FUNCTION_BLOCK FB_ServoVise
VAR_INPUT
	bErrorAck				: BOOL;
	bEnable					: BOOL;
	eCommand				: E_ServoVise_Command;
	bManualMode				: BOOL;
	lrTargetDistance		: LREAL;			// [mm]		Target distance without torque limit
	lrVisePosition			: LREAL;			// [mm]		Value of distance sensor
	bVisePosValid			: BOOL;				// []		Distane sensor status
	nTargetVelocity			: LREAL;			// [mm/s]
	nTorque					: LREAL := 20.0;	// [Nm]
	nTorqueRamp				: LREAL := 10.0;	// [%/s]
	nTorqueVelocityLimit	: LREAL := 0.1;		// [mm/s]
	nOverride				: LREAL := 100.0;	// [%] 
	nAttachVelocity			: LREAL := 0.1;
	nCalOffset_1			: LREAL := 22.32;
	nCalOffset_2			: LREAL := 99.01;
	nOpenOffset				: LREAL := 4;
	eViseJawState			: E_ViseJawState := E_ViseJawState.P1_0_120;
	stAxisEvent				: TcEventEntry;	(*Event definition*)
END_VAR
VAR_OUTPUT
	bReady					: BOOL;
	bBusy 					: BOOL;
	bDone 					: BOOL;
	bError 					: BOOL;
END_VAR
VAR (* Drive *)
	Axis					: AXIS_REF;
	fbPower					: MC_Power;
	fbMoveRelative			: MC_MoveRelative;
	fbReadDriveOpMode		: MC_ReadDriveOperationMode;
	fbWriteDriveOpMode		: MC_WriteDriveOperationMode;
	fbStop					: MC_Halt;
	fbHalt					: MC_Stop;
	fbTorqueControl			: MC_TorqueControl;	
	fbJog					: MC_Jog;
	fbTorqueCheck			: FB_TorqueCheck;	

	fbSoEReset				: FB_SoEReset;
	fbReset					: MC_Reset;
END_VAR
VAR (* State control *)
	nState 					: UDINT;
	nLastState				: UDINT;
	sState					: STRING;
	nTorqueRelief			: LREAL := 0.005;	// 0.005mm = 0.9°
	
	// Error control
	bIsInitalized			: BOOL;
	fbAlarm					: FB_TcAlarm;
	nGlobalAxisErrorID		: UDINT;
	
	//LastStates
	anLastStates			: ARRAY[0..500] OF UDINT;
    iLastStates				: INT;
	nRealVisePos			: LREAL;
END_VAR
VAR CONSTANT									//																			%     Tmax    i   Theta															
	nTScale					: LREAL := 2.3923;	// nTorque[Nm] / nTScale[Nm/%] = Required_torque_value[%]		{nTScale = 0.01 * 5.09 * 50 * 0.94}
END_VAR

(* Timers **************************************)

(* Enable **************************************)
IF NOT bEnable THEN
	fbPower.Enable := FALSE;
	fbTorqueControl.Execute := FALSE;
	fbMoveRelative.Execute := FALSE;
	nState := 0;
END_IF

(* States **************************************)
IF nLastState <> nState THEN
	nLastState := nState;
END_IF

(* State history ************************************************)
IF(nState >= 100) AND (nState <= 20000) THEN
(*Steps before any state*)
	IF anLastStates[0] <> nState THEN
		FOR iLastStates:=500 TO 1 BY -1 DO
			anLastStates[iLastStates]:= anLastStates[iLastStates-1];
		END_FOR
		anLastStates[0]:= nState;
	END_IF
END_IF	

(* Manual mode **************************************)
IF bManualMode THEN
	nState := 150000;
END_IF

(*Calculate Vise position **************************************)
IF eViseJawState = E_ViseJawState.P1_0_120 THEN
	nRealVisePos := lrVisePosition + nCalOffset_1;
ELSE
	nRealVisePos := lrVisePosition + nCalOffset_2;
END_IF

(* Error handling Tc3_EventLogger *******************************)
IF NOT bIsInitalized THEN
	bIsInitalized  :=  TRUE;
	fbAlarm.CreateEx(stAxisEvent, TRUE, 0);
END_IF

(* Error acknoledge **************************************)
IF bErrorAck THEN
	IF fbAlarm.eConfirmationState = 2 THEN
		fbAlarm.Confirm(0);
	END_IF
END_IF

IF Axis.Status.Error OR Axis.Status.DriveDeviceError OR fbPower.Error OR fbMoveRelative.Error OR fbTorqueControl.Error OR
	fbJog.Error OR fbSoEReset.Error OR fbReset.Error OR fbHalt.Error OR fbStop.Error OR fbReadDriveOpMode.Error OR fbWriteDriveOpMode.Error
THEN
	bError  :=  TRUE;
	IF (fbAlarm.eConfirmationState <> 2 AND fbAlarm.nTimeCleared <> 0 AND fbAlarm.nTimeConfirmed <> 0) OR //Ha már volt alarm, akkor van bennük érték
		(fbAlarm.eConfirmationState = 1 AND fbAlarm.nTimeCleared = 0 AND fbAlarm.nTimeConfirmed = 0)	//Első futás esetén
	THEN
		//fb_DriveDiag(Execute :=  TRUE, Axis :=  Axis);
		//IF NOT fb_DriveDiag.Busy THEN
			//fb_DriveDiag(Execute :=  FALSE, Axis :=  Axis);
			IF Axis.Status.ErrorID <> 0 THEN
				nGlobalAxisErrorID  :=  Axis.Status.ErrorID;
			ELSIF fbPower.ErrorID <> 0 THEN
				nGlobalAxisErrorID  :=  fbPower.ErrorID;
			ELSIF fbMoveRelative.ErrorID <> 0 THEN
				nGlobalAxisErrorID  :=  fbMoveRelative.ErrorID;
			ELSIF fbTorqueControl.ErrorID <> 0 THEN
				nGlobalAxisErrorID  :=  fbTorqueControl.ErrorID;
			ELSIF fbJog.ErrorID <> 0 THEN
				nGlobalAxisErrorID  :=  fbJog.ErrorID;
			ELSIF fbSoEReset.SercosErrId <> 0 THEN
				nGlobalAxisErrorID  :=  fbSoEReset.SercosErrId;
			ELSIF fbReset.ErrorID <> 0 THEN
				nGlobalAxisErrorID  :=  fbReset.ErrorID;
			END_IF
			//fbAlarm.ipArguments.Clear().AddUDInt(nGlobalAxisErrorID).AddUDInt(fb_DriveDiag.DiagNumber);
			fbAlarm.ipArguments.Clear().AddUDInt(nGlobalAxisErrorID);
			fbAlarm.Raise(0);
		//END_IF
	END_IF
END_IF

Axis();

CASE nState OF
{region "Alaphelyzet felvétel"}
	(****************************************************************************************)
	(******************************* Alaphelyzetfelvétel ************************************)
	(****************************************************************************************)	
	0:		(*-----=== Kimenetek törlése ===-----*)
		fbPower.Enable := FALSE;
		fbReadDriveOpMode.Execute := FALSE;
		fbWriteDriveOpMode.Execute := FALSE;
		fbStop.Execute := FALSE;
		fbHalt.Execute := FALSE;
		fbTorqueControl.Execute := FALSE;
		fbMoveRelative.Execute := FALSE;
		bBusy := FALSE;
		bDone := FALSE;
		bError := FALSE;
		IF bEnable THEN
			nState := nState + 20;
		END_IF
		
	20:		(*-----=== Axis és Drive hibák ellenőrzése ===-----*)
		IF Axis.Status.Error OR Axis.Status.DriveDeviceError THEN
			nState := 250000;
		ELSIF bEnable THEN
			nState := nState + 20;
		END_IF

	40:		(*-----=== Drive Op. mód ellenörzés ===-----*)
		fbReadDriveOpMode.Execute := TRUE;
		IF fbReadDriveOpMode.Done THEN
			IF fbReadDriveOpMode.DriveOperationMode <> Tc2_MC2.E_DriveOperationMode.DriveOperationMode_Default THEN
				nState := 10000;
			ELSE
				nState := 100;
			END_IF
			fbReadDriveOpMode.Execute := FALSE;
		END_IF

	100:		(*-----=== Drive átkapcsolása PtP módba ===-----*)
		fbWriteDriveOpMode.DriveOperationMode := Tc2_MC2.E_DriveOperationMode.DriveOperationMode_Default;
		fbWriteDriveOpMode.Execute := TRUE;
		IF fbWriteDriveOpMode.Done THEN
			fbWriteDriveOpMode.Execute := FALSE;
			nState := 10000;
		END_IF
{endregion}

{region "Alaphelyzet"}
	(****************************************************************************************)
	(*********************************** Alaphelyzet ****************************************)
	(****************************************************************************************)	
	10000:		(*-----=== Várakozás parancsra ===-----*)
		bReady := TRUE;
		bBusy := FALSE;
		bDone := FALSE;
		IF eCommand = E_ServoVise_Command.Fix THEN				// Nyomatékra húzás
			bBusy := TRUE;
			nState := 20000;
		ELSIF eCommand = E_ServoVise_Command.MoveToPos THEN		// Pozícionálás
			bBusy := TRUE;
			nState := 40000;
		ELSIF eCommand = E_ServoVise_Command.Release THEN		// Kioldás
			bBusy := TRUE;
			nState := 60000;
		ELSIF eCommand = E_ServoVise_Command.Attach THEN		// Tengelykapcsoló csatlakoztatása
			bBusy := TRUE;
			nState := 80000;
		END_IF
{endregion}

{region "Satu nyomatékrahúzása"}
	(****************************************************************************************)
	(****************************** Satu nyomatékrahúzás ************************************)
	(****************************************************************************************)	
	20000:		(*-----=== Szervo BE ===-----*)
		fbPower.Enable := TRUE;
		IF fbPower.Status THEN
			nState := 20100;
		ELSIF fbPower.Error THEN
			IF bStepEnable THEN
				nState := 250000;
			END_IF
		END_IF	
		
	20100:		(*-----=== Zárás nyomatékra ===-----*)
		fbTorqueControl.Torque := -1 * ABS(nTorque/nTScale);					// Nyomaték átszámítása Nm-ből %-ba
		fbTorqueControl.TorqueRamp := nTorqueRamp;
		fbTorqueControl.VelocityLimitHigh := nTorqueVelocityLimit;
		fbTorqueControl.VelocityLimitLow := -1 * nTorqueVelocityLimit;
		fbTorqueControl.Execute := TRUE;
		IF fbTorqueControl.Busy THEN
			IF bStepEnable THEN
				nTorqueRelief := ((ABS(nTorque))/6000 + (1/300));					// A feszültségmentesítési szög nyomatékfüggő!! Y=m*X+b	{m=1/6000, b=1/300}
				nState := nState + 20;
			END_IF
		END_IF
	
	20120:		(*-----=== Nyomaték figyelés ===-----*)
		IF fbTorqueCheck.bTorqueDone THEN
			IF bStepEnable THEN
				fbTorqueControl.Execute := FALSE;
				nState := nState + 20;
			END_IF
		ELSIF fbTorqueControl.Error THEN
			nState := 250000;
		ELSIF (lrVisePosition < 0) AND bVisePosValid THEN						// Minimális pozíció elérve -> Hiba
			nState := 250000;
		ELSIF (nRealVisePos < (lrTargetDistance - 4)) THEN						// Satupozíció 4mm-el kissebb mint a nominál méret -> Hiba
			nState := 250000;
		END_IF	
	
	20140:		(*-----=== Axis Halt ===-----*)(*-----=== Váratla mozgások elkerülése ===-----*)
		fbHalt.Execute := TRUE;
		IF fbHalt.Done THEN
			IF bStepEnable THEN
				fbHalt.Execute := FALSE;
				nState:= nState + 20;
			END_IF
		END_IF
	
	20160:		(*-----=== Átkapcsolás pozíció módba ===-----*)
		fbWriteDriveOpMode.DriveOperationMode := Tc2_MC2.E_DriveOperationMode.DriveOperationMode_Default;
		fbWriteDriveOpMode.Execute := TRUE;
		IF fbWriteDriveOpMode.Done THEN
			IF bStepEnable THEN
				fbWriteDriveOpMode.Execute := FALSE;
				nState := nState + 20;
			END_IF
		END_IF
	
	20180:		(*-----=== Szervo Mozgatás PtP ===-----*)
		fbMoveRelative.Distance := nTorqueRelief;
		fbMoveRelative.Velocity := nTargetVelocity;
		fbMoveRelative.Execute := TRUE;
		IF fbMoveRelative.Done THEN
			IF bStepEnable THEN
				fbMoveRelative.Execute := FALSE;
				nState := nState + 20;
			END_IF
		ELSIF fbMoveRelative.Error THEN
			fbMoveRelative.Execute := FALSE;
			nState := 250000;
		END_IF
	
	20200:		(*-----=== Szervo KI ===-----*)
		fbPower.Enable := FALSE;
		nState := nState + 20;
	
	20220:		(*-----=== Várakozás parancs törlésre ===-----*)
		bBusy := FALSE;
		bDone := TRUE;
		IF eCommand = E_ServoVise_Command.NoCommand THEN
			IF bStepEnable THEN
				nState := 10000;
			END_IF
		END_IF
{endregion}

{region "Satu pzícionálás"}
	(****************************************************************************************)
	(********************************* Satu pozícionálás ************************************)
	(****************************************************************************************)	
	40000:		(*-----=== Szervo BE ===-----*)
		fbPower.Enable := TRUE;
		IF fbPower.Status THEN
			nState := nState + 20;
		ELSIF fbPower.Error THEN
			nState := 250000;
		END_IF
			
	40020:		(*-----=== Szervo Mozgatás PtP ===-----*)
		fbMoveRelative.Distance := (lrTargetDistance + nOpenOffset) - nRealVisePos;
		fbMoveRelative.Velocity := nTargetVelocity;
		fbMoveRelative.Execute := TRUE;
		IF fbMoveRelative.Done THEN
			IF bStepEnable THEN
				fbMoveRelative.Execute := FALSE;
				nState := nState + 20;
			END_IF
		ELSIF fbMoveRelative.Error THEN
			fbMoveRelative.Execute := FALSE;
			nState := 250000;
		ELSIF (lrVisePosition < 0) AND bVisePosValid THEN						// Minimális pozíció elérve -> Hiba
			nState := 250000;
		ELSIF (nRealVisePos < (lrTargetDistance - 4)) THEN						// Satupozíció 4mm-el kissebb mint a nominál méret -> Hiba
			nState := 250000;
		END_IF
		
	40040:		(*-----=== Szervo KI ===-----*)
		fbPower.Enable := FALSE;
		nState := nState + 20;
	
	40060:		(*-----=== Várakozás parancs törlésre ===-----*)
		bBusy := FALSE;
		bDone := TRUE;
		IF eCommand = E_ServoVise_Command.NoCommand THEN
			IF bStepEnable THEN
				nState := 10000;
			END_IF
		END_IF
{endregion}

{region "Satu oldása"}
	(****************************************************************************************)
	(************************************ Satu elengedés ************************************)
	(****************************************************************************************)
	60000:		(*-----=== Szervo BE ===-----*)
		fbPower.Enable := TRUE;
		IF fbPower.Status THEN
			nState := nState + 20;
		ELSIF fbPower.Error THEN
			nState := 250000;
		END_IF
	
	60020:		(*-----=== Szervo Mozgatás PtP ===-----*)
		fbMoveRelative.Distance := nOpenOffset;
		fbMoveRelative.Velocity := nTargetVelocity;
		fbMoveRelative.Execute := TRUE;
		IF fbMoveRelative.Done THEN
			IF bStepEnable THEN
				fbMoveRelative.Execute := FALSE;
				nState := nState + 20;
			END_IF
		ELSIF fbMoveRelative.Error THEN
			fbMoveRelative.Execute := FALSE;
			nState := 250000;
		END_IF
	
	60040:		(*-----=== Szervo KI ===-----*)
		fbPower.Enable := FALSE;
		nState := nState + 20;
		
	60060:		(*-----=== Várakozás parancs törlésre ===-----*)
		bBusy := FALSE;
		bDone := TRUE;
		IF eCommand = E_ServoVise_Command.NoCommand THEN
			IF bStepEnable THEN
				nState := 10000;
			END_IF
		END_IF
{endregion}

{region "Satu csatlakoztatása"}
	(****************************************************************************************)
	(********************************** Satu csatlakoztatás *********************************)
	(****************************************************************************************)
	80000:		(*-----=== Szervo BE ===-----*)
		fbPower.Enable := TRUE;
		IF fbPower.Status THEN
			nState := nState + 20;
		ELSIF fbPower.Error THEN
			nState := 250000;
		END_IF	
		
	80020:		(*-----=== Zárás nyomatékra ===-----*)
		fbTorqueControl.Torque := -5;
		fbTorqueControl.TorqueRamp := nTorqueRamp;
		fbTorqueControl.VelocityLimitHigh := nAttachVelocity;
		fbTorqueControl.VelocityLimitLow := -1 * nAttachVelocity;
		fbTorqueControl.Execute := TRUE;
		IF fbTorqueControl.Busy THEN
			IF bStepEnable THEN
				nState := nState + 20;
			END_IF
		END_IF
	
	80040:		(*-----=== Várakozás parancs törlésre ===-----*)
		bBusy := FALSE;
		bDone := TRUE;
		IF eCommand = E_ServoVise_Command.NoCommand THEN
			IF bStepEnable THEN
				fbTorqueControl.Execute := FALSE;
				nState:= nState + 20;
			END_IF
		END_IF
	
	80060:		(*-----=== Axis Halt ===-----*)(*-----=== Váratla mozgások elkerülése ===-----*)
		fbHalt.Execute := TRUE;
		IF fbHalt.Done THEN
			IF bStepEnable THEN
				fbHalt.Execute := FALSE;
				nState:= nState + 20;
			END_IF
		END_IF
	
	80080:		(*-----=== Átkapcsolás pozíció módba ===-----*)
		fbWriteDriveOpMode.DriveOperationMode := Tc2_MC2.E_DriveOperationMode.DriveOperationMode_Default;
		fbWriteDriveOpMode.Execute := TRUE;
		IF fbWriteDriveOpMode.Done THEN
			IF bStepEnable THEN
				fbWriteDriveOpMode.Execute := FALSE;
				nState := nState + 20;
			END_IF
		END_IF
	
	80100:		(*-----=== Szervo KI ===-----*)
		fbPower.Enable := FALSE;
		nState := 10000;
{endregion}

{region "Manual mód"}
	(****************************************************************************************)
	(*************************************** Kézi üzem **************************************)
	(****************************************************************************************)	
	150000:		(*-----=== Manual mode ===-----*)
		fbJog.Mode := MC_JOGMODE_CONTINOUS;
		IF NOT bManualMode THEN
			nState := 10000;
		END_IF
		IF fbJog.Error THEN
			nState := 250000;
		END_IF
{endregion}

{region "Hibakezelés"}
	(****************************************************************************************)
	(************************************* Hibakezelés **************************************)
	(****************************************************************************************)	
	250000:		(*-----=== Error ===-----*)
		bReady := FALSE;
		bBusy := FALSE;
		bDone := FALSE;
		bError := TRUE;
		fbReadDriveOpMode.Execute := FALSE;
		fbWriteDriveOpMode.Execute := FALSE;
		fbStop.Execute := FALSE;
		fbHalt.Execute := FALSE;
		fbTorqueControl.Execute := FALSE;
		fbMoveRelative.Execute := FALSE;
		IF Axis.Status.HasJob THEN
			nState := nState + 20;
		ELSE
			nState := nState + 40;
		END_IF
	
	250020:	(* Axis halt *)
		fbHalt.Execute := TRUE;
		IF fbHalt.Done THEN
			IF bStepEnable THEN
				fbHalt.Execute := FALSE;
				nState:= nState + 20;
			END_IF
		END_IF
	
	250040: (*Wait error ACK*)
		IF bErrorAck THEN
			nState := nState + 20;
		END_IF
		
	250060: (*Error ACK*)
		IF Axis.Status.DriveDeviceError THEN
			IF bStepEnable THEN 
				fbSoEReset.Execute := TRUE;
				fbReset.Execute := TRUE;
				nState := 250080;
			END_IF
		ELSIF Axis.Status.Error THEN
			IF bStepEnable THEN 
				fbReset.Execute := TRUE;
				nState := 250100;
			END_IF
		ELSE
			nState := 0;
		END_IF
		
	250080: (*Drive Reset*)
		IF NOT fbSoEReset.Busy THEN
			fbSoEReset.Execute := FALSE;
			nState := 0;
		ELSIF fbSoEReset.Error THEN
			nState := 0; 
		END_IF
		
	250100: (*Reset*)
		IF fbReset.Done THEN
			fbReset.Execute := FALSE;
			nState := 0;
		ELSIF fbReset.Error THEN
			nState := 0; 
		END_IF	
{endregion}
ELSE
	sState := 'Not used step';	
END_CASE


ActPower();
ActHalt();
ActStop();
ActMode();
ActTorque();
ActMoveRelative();
ActJog();
ActSoEReset();
ActReset();

ACTION ActHalt:
fbHalt(Axis:= Axis);
END_ACTION

ACTION ActJog:
fbJog(
	Axis:= Axis, 
	JogForward:= TRUE, 
	JogBackwards:= TRUE, 
	Mode:= fbJog.Mode, 
	Velocity:= 10);
END_ACTION

ACTION ActMode:
fbReadDriveOpMode(
	Axis:= Axis, 
	Execute:= , 
	Options:= , 
	Done=> , 
	Busy=> , 
	Error=> , 
	ErrorID=> , 
	DriveOperationMode=> );

fbWriteDriveOpMode(
	Axis:= Axis, 
	Execute:= , 
	DriveOperationMode:= , 
	Options:= , 
	Done=> , 
	Busy=> , 
	Error=> , 
	ErrorID=> );
END_ACTION

ACTION ActMoveRelative:
fbMoveRelative(
	Axis:= Axis);
//, 
//	Distance:= lrCalculatedDistance, 
//	Velocity:= nOpenVelocity);
END_ACTION

ACTION ActPower:
fbPower(
	Axis:= Axis, 
	Enable_Positive:= TRUE, 
	Enable_Negative:= TRUE, 
	Override:= nOverride);
END_ACTION

ACTION ActReset:
fbReset(Axis:= Axis);
END_ACTION

ACTION ActSoEReset:
fbSoEReset(Axis:= Axis);
END_ACTION

ACTION ActStop:
fbStop(Axis:= Axis);
END_ACTION

ACTION ActTorque:
fbTorqueControl(
	Axis:= Axis, 
	ContinuousUpdate:= FALSE, 
	Relative:= FALSE, 
	Torque:= , 
	TorqueRamp:= , 
	VelocityLimitHigh:= , 
	VelocityLimitLow:= );

fbTorqueCheck(
	Axis:= Axis, 
	bEnable:= fbTorqueControl.Execute, 
	nTorque:= fbTorqueControl.Torque, 
	tTorqueStabTime:= T#500ms, 
	bTorqueDone=> );
END_ACTION

END_FUNCTION_BLOCK

(* stored: Version 1.1.0.1, ProductVersion 3.1.4024.12
   POU FB_ServoVise: Id {6aa55fe7-afee-4b40-bb31-d2de59dbb683}, SpecialFunc None
   Action ActHalt: Id {e3aaa0fe-3cea-4fea-a021-0bd63a7bcba7}
   Action ActJog: Id {dbec480c-3b95-4842-b96d-a3a6b738e551}
   Action ActMode: Id {f8ae5c0a-b76d-4cf9-8294-fc8ed7f21ff5}
   Action ActMoveRelative: Id {faed1f2c-59cc-4df3-b558-77214563147a}
   Action ActPower: Id {dab1f324-c7df-460d-9b39-6efd4ef1e589}
   Action ActReset: Id {f8efa3f5-5e55-468b-af9d-9a506b6e8629}
   Action ActSoEReset: Id {ee4f3b79-5d36-4fe1-8e3a-25aa07755642}
   Action ActStop: Id {f39d1764-a57b-4254-8962-1c3d4265c9c5}
   Action ActTorque: Id {d2bf8c67-a3a8-41bb-99a1-1ee7a27893c3} *)
